// TIA Portal V18 export
ORGANIZATION_BLOCK "Main"   // OB1, LAD, ProgramCycle
TITLE = "Main Program Sweep (Cycle)"
{ S7_Optimized_Access := 'TRUE' }
VERSION : 0.1
// stored: AutoNumber true, IsIECCheckEnabled false, SetENOAutomatically false
   VAR_INPUT
      Initial_Call : Bool;   // Initial call of this OB
      Remanence : Bool;   // =True, if remanent data are available
   END_VAR
BEGIN

REGION Network 1
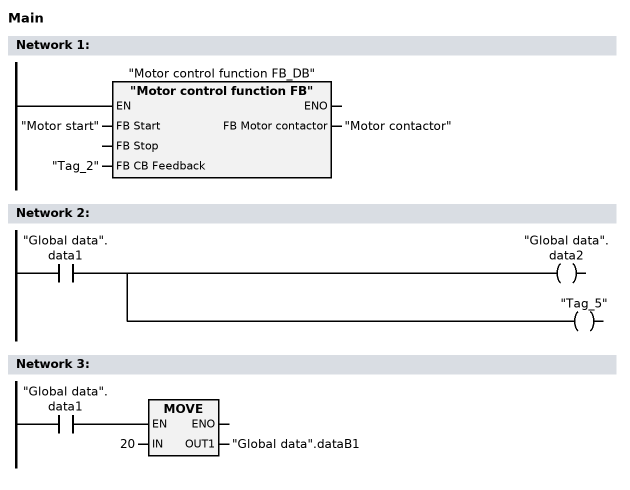
   RUNG wire#powerrail
      "Motor control function FB_DB"("FB Start" := "Motor start", "FB Stop" :=, "FB CB Feedback" := "Tag_2", "FB Motor contactor" => "Motor contactor")
   END_RUNG
   // the same network as SCL:
   "Motor control function FB_DB"("FB Start" := "Motor start",   // "Motor control function FB"
                           "FB CB Feedback" := "Tag_2",
                           "FB Motor contactor" => "Motor contactor");
END_REGION

REGION Network 2
   RUNG wire#powerrail
      Contact( "Global data".data1 )
      wire#w1
      Coil( "Global data".data2 )
   END_RUNG
   RUNG wire#w1
      Coil( "Tag_5" )
   END_RUNG
   // the same network as SCL:
   "Global data".data2 := "Global data".data1;
   "Tag_5" := "Global data".data1;
END_REGION

REGION Network 3
   RUNG wire#powerrail
      Contact( "Global data".data1 )
      Move(in := 20, out1 => "Global data".dataB1)
   END_RUNG
   // the same network as SCL:
   IF "Global data".data1 THEN "Global data".dataB1 := 20; END_IF;
END_REGION
END_ORGANIZATION_BLOCK
